(* IEC 61131-3 sources: InfiniteStateMachine/extracted_st/infinitestatemachine/function_blocks/statemachine/enter, 1 file *)

(* ---- Enter.st ---- *)
(* --- Interface --- *)
METHOD PROTECTED Enter
VAR_INPUT
	itfState : IState;
END_VAR

(* --- Implementation --- *)
IF Push(itfState) THEN
	itfState.Enter(THIS^);
END_IF
